// TIA Portal V16 export
// export: Created 2022-04-14T22:38:29.5961786Z, ExportSetting WithDefaults, DisplayName Totally Integrated Automation Portal, DisplayVersion V16, DisplayName TIA Portal Version Control Interface, DisplayVersion V16, DisplayName TIA Portal Openness, DisplayVersion V16, DisplayName STEP 7 Professional, DisplayVersion V16, DisplayName STEP 7 Safety, DisplayVersion V16, DisplayName WinCC Professional, DisplayVersion V16
FUNCTION_BLOCK "04 Count"   // FB4, LAD
{ S7_Optimized_Access := 'TRUE' }
VERSION : 0.1
// stored: AutoNumber true, IsIECCheckEnabled false, IsRetainMemResEnabled false, MemoryReserve 100, SetENOAutomatically false, UDAEnableTagReadback false
   VAR_TEMP   // added for the SCL form of the ladder/FBD networks
      _w1 : Bool;
      _w2 : Bool;
      _w3 : Bool;
   END_VAR
BEGIN

REGION Network 1: Items count
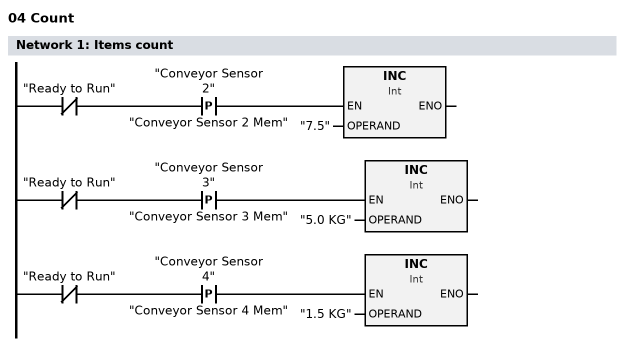
   RUNG wire#powerrail
      I_Contact( "Ready to Run" )
      P_Contact(operand := "Conveyor Sensor 2", bit := "Conveyor Sensor 2 Mem")
      { S7_Templates := "DestType := Int" } Inc( "7.5" )
   END_RUNG
   RUNG wire#powerrail
      I_Contact( "Ready to Run" )
      P_Contact(operand := "Conveyor Sensor 3", bit := "Conveyor Sensor 3 Mem")
      { S7_Templates := "DestType := Int" } Inc( "5.0 KG" )
   END_RUNG
   RUNG wire#powerrail
      I_Contact( "Ready to Run" )
      P_Contact(operand := "Conveyor Sensor 4", bit := "Conveyor Sensor 4 Mem")
      { S7_Templates := "DestType := Int" } Inc( "1.5 KG" )
   END_RUNG
   // the same network as SCL:
   #_w1 := NOT "Ready to Run" AND "Conveyor Sensor 2" AND NOT "Conveyor Sensor 2 Mem";   // rising edge of "Conveyor Sensor 2"
   "Conveyor Sensor 2 Mem" := "Conveyor Sensor 2";
   IF #_w1 THEN "7.5" := "7.5" + 1; END_IF;
   #_w2 := NOT "Ready to Run" AND "Conveyor Sensor 3" AND NOT "Conveyor Sensor 3 Mem";   // rising edge of "Conveyor Sensor 3"
   "Conveyor Sensor 3 Mem" := "Conveyor Sensor 3";
   IF #_w2 THEN "5.0 KG" := "5.0 KG" + 1; END_IF;
   #_w3 := NOT "Ready to Run" AND "Conveyor Sensor 4" AND NOT "Conveyor Sensor 4 Mem";   // rising edge of "Conveyor Sensor 4"
   "Conveyor Sensor 4 Mem" := "Conveyor Sensor 4";
   IF #_w3 THEN "1.5 KG" := "1.5 KG" + 1; END_IF;
END_REGION
END_FUNCTION_BLOCK
